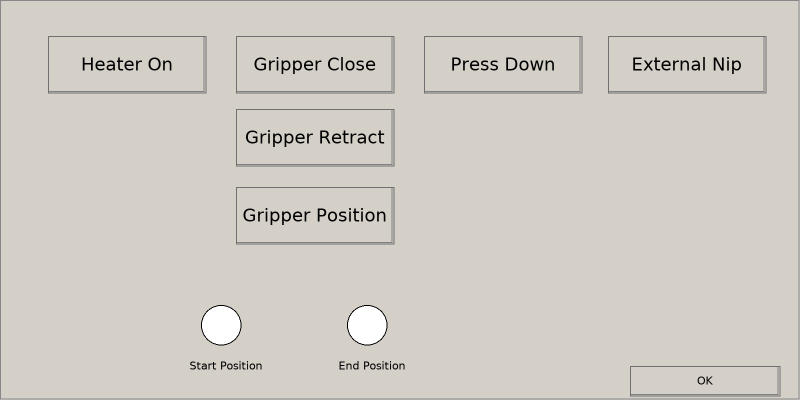
VISUALIZATION Dialog_IO  // 800x400
    Button (48,36 158x57), "Heater On"
        toggle gMachineCtrl.IO.Out.HeaterOn
    Button (236,36 158x57), "Gripper Close"
        toggle gMachineCtrl.IO.Out.GripperOpen
    Button (236,109 158x57), "Gripper Retract"
        toggle gMachineCtrl.IO.Out.GripperRetract
    Button (236,187 158x57), "Gripper Position"
        toggle gMachineCtrl.IO.Out.GripperPistonPosition
    Button (424,36 158x57), "Press Down"
        toggle gMachineCtrl.IO.Out.PressDown
    Button (630,366 150x30), "OK"
        OnMouseDown: CloseDialog Dialog=Dialog_IO, Result=OK, NumpadKeypadSet=True
    Button (608,36 158x57), "External Nip"
        toggle gMachineCtrl.IO.Out.ExternalNipMotor
    Ellipse (201,305 40x40), colour toggle: gMachineCtrl.IO.In.GripperStartPosition
    Label (171,351 110x30), "Start Position"
    Ellipse (347,305 40x40), colour toggle: gMachineCtrl.IO.In.GripperStartPosition
    Label (317,351 110x30), "End Position"
END_VISUALIZATION

(* stored: Version 1.1.0.1, ProductVersion 3.1.4024.3
   Visu Dialog_IO: Id {9c8c5e7e-3a95-406b-accf-bd5546b5fed8} *)
